FUNCTION_BLOCK DigitalController
  (* Standard: 61499-2 *)
  (* Version 0.1, 2015-00-11, syy, syy-PC *)
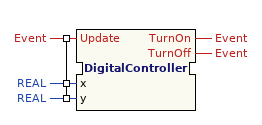
  EVENT_INPUT
    Update WITH x, y;
  END_EVENT
  EVENT_OUTPUT
    TurnOn;
    TurnOff;
  END_EVENT
  VAR_INPUT
    x : REAL;
    y : REAL;
  END_VAR
  VAR
    control : REAL;
    timer : REAL;
  END_VAR
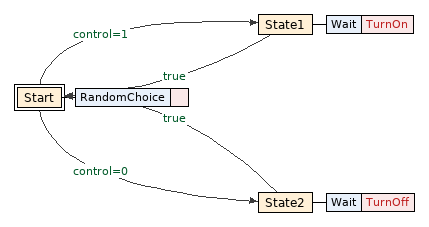
  EC_STATES
    Start : RandomChoice;
    State1 : Wait -> TurnOn;
    State2 : Wait -> TurnOff;
  END_STATES
  EC_TRANSITIONS
    Start TO State1 := control=1;
    Start TO State2 := control=0;
    State1 TO Start := true;
    State2 TO Start := true;
  END_TRANSITIONS
  ALGORITHM RandomChoice IN C:
me->timer=0;

/* Intializes random number generator */
srand(time(NULL));

me->control = rand() % 2 ;
//printf("control : %d\n", me->control);
  END_ALGORITHM
  ALGORITHM Wait IN C:
//printf("signal sent\n");
wait(10);
//me->timer++;
  END_ALGORITHM
END_FUNCTION_BLOCK
